SUBAPPLICATION Uebung_083 (* Beispiel für E_CTUD_UDINT *)
  (* Standard: 61499-2; Description: Beispiel für E_CTD Aufwärts zählen UAO Curriculum Module 3 - The IEC 61499 Standard, Seite 94 *)
  (* Version 1.0, 2023-10-23, franz *)
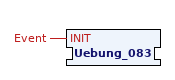
  EVENT_INPUT
    INIT;
  END_EVENT
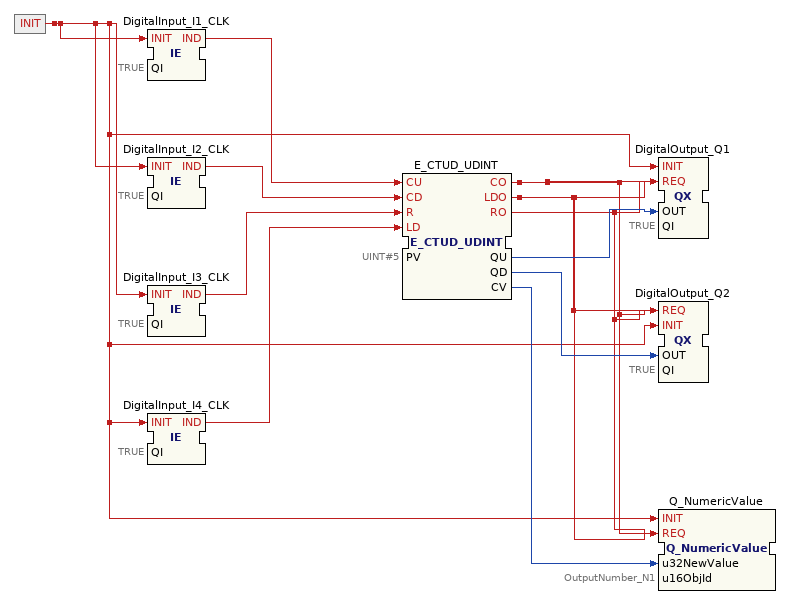
  FBS
    DigitalOutput_Q1 : QX(QI := TRUE);
    DigitalInput_I1_CLK : IE(QI := TRUE);
    E_CTUD_UDINT : E_CTUD_UDINT(PV := UINT#5);
    DigitalInput_I2_CLK : IE(QI := TRUE);
    DigitalInput_I3_CLK : IE(QI := TRUE);
    DigitalInput_I4_CLK : IE(QI := TRUE);
    DigitalOutput_Q2 : QX(QI := TRUE);
    Q_NumericValue : Q_NumericValue(u16ObjId := OutputNumber_N1);
  END_FBS
  EVENT_CONNECTIONS
    INIT TO DigitalInput_I1_CLK.INIT;
    INIT TO DigitalOutput_Q1.INIT;
    DigitalInput_I1_CLK.IND TO E_CTUD_UDINT.CU;
    E_CTUD_UDINT.CO TO DigitalOutput_Q1.REQ;
    E_CTUD_UDINT.LDO TO DigitalOutput_Q1.REQ;
    INIT TO DigitalInput_I2_CLK.INIT;
    DigitalInput_I2_CLK.IND TO E_CTUD_UDINT.CD;
    E_CTUD_UDINT.RO TO DigitalOutput_Q1.REQ;
    INIT TO DigitalInput_I3_CLK.INIT;
    DigitalInput_I3_CLK.IND TO E_CTUD_UDINT.R;
    INIT TO DigitalInput_I4_CLK.INIT;
    DigitalInput_I4_CLK.IND TO E_CTUD_UDINT.LD;
    E_CTUD_UDINT.LDO TO DigitalOutput_Q2.REQ;
    INIT TO DigitalOutput_Q2.INIT;
    E_CTUD_UDINT.CO TO DigitalOutput_Q2.REQ;
    E_CTUD_UDINT.RO TO DigitalOutput_Q2.REQ;
    INIT TO Q_NumericValue.INIT;
    E_CTUD_UDINT.CO TO Q_NumericValue.REQ;
    E_CTUD_UDINT.RO TO Q_NumericValue.REQ;
    E_CTUD_UDINT.LDO TO Q_NumericValue.REQ;
  END_CONNECTIONS
  DATA_CONNECTIONS
    E_CTUD_UDINT.QU TO DigitalOutput_Q1.OUT;
    E_CTUD_UDINT.QD TO DigitalOutput_Q2.OUT;
    E_CTUD_UDINT.CV TO Q_NumericValue.u32NewValue;
  END_CONNECTIONS
END_SUBAPPLICATION
